// Mitsubishi GX Works2 project: 서보 모터 정보 복붙용   PLC: Q03UDV

PROGRAM MAIN
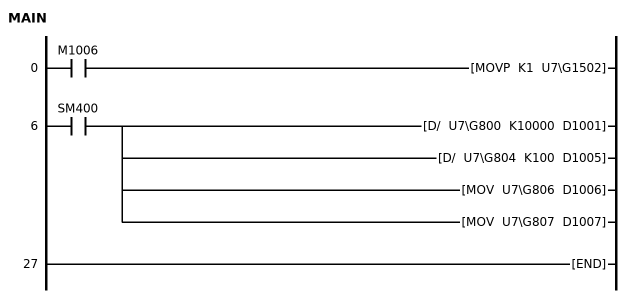
0     LD      M1006
      MOVP    K1 U7\G1502
6     LD      SM400
      D/      U7\G800 K10000 D1001
      D/      U7\G804 K100 D1005
      MOV     U7\G806 D1006
      MOV     U7\G807 D1007
27    END
END_PROGRAM
